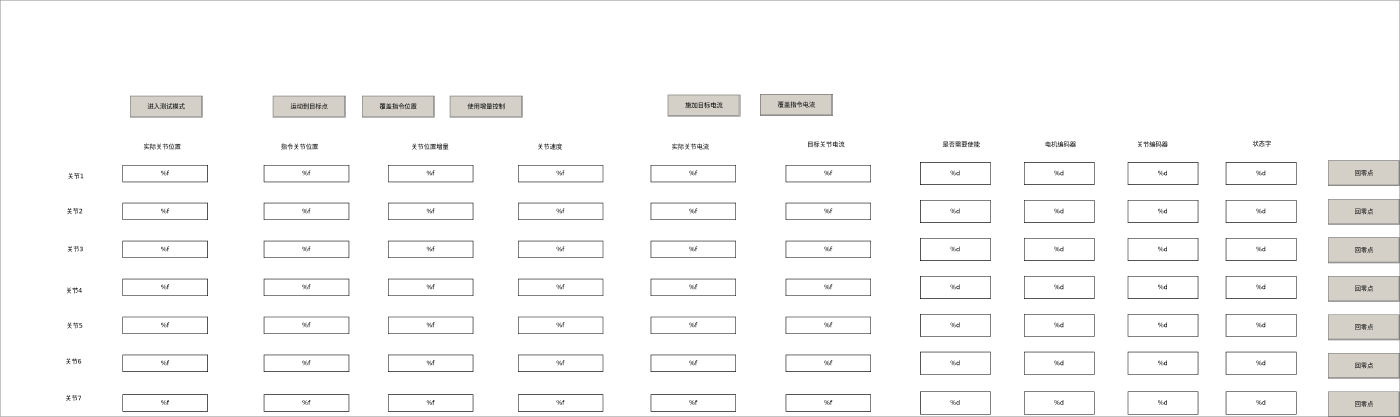
VISUALIZATION motion_a2  // 2468x736
    Label (211,244 150x30), "实际关节位置"
    Rectangle (216,291 150x30), "%f", text variable: g_motionTest.m_armDHJntPos[2][1]
    Label (453,244 150x30), "指令关节位置"
    Label (683,244 150x30), "关节位置增量"
    Rectangle (684,291 150x30), "%f", text variable: g_motionTest.m_targetJntPosInc[2][1]
        OnMouseClick: write the text variable via Default
    Label (1142,244 150x30), "实际关节电流"
    Rectangle (1147,291 150x30), "%f", text variable: g_motionTest.m_curJntCurrent[2][1]
    Label (1381,240 150x30), "目标关节电流"
    Rectangle (1385,291 150x30), "%f", text variable: g_motionTest.m_targetJntCurrent[2][1]
        OnMouseClick: write the text variable via Default
    Rectangle (216,358 150x30), "%f", text variable: g_motionTest.m_armDHJntPos[2][2]
    Rectangle (216,425 150x30), "%f", text variable: g_motionTest.m_armDHJntPos[2][3]
    Rectangle (216,492 150x30), "%f", text variable: g_motionTest.m_armDHJntPos[2][4]
    Rectangle (216,559 150x30), "%f", text variable: g_motionTest.m_armDHJntPos[2][5]
    Rectangle (216,626 150x30), "%f", text variable: g_motionTest.m_armDHJntPos[2][6]
    Rectangle (216,696 150x30), "%f", text variable: g_motionTest.m_armDHJntPos[2][7]
    Rectangle (465,291 150x30), "%f", text variable: g_motionTest.m_targetJntPos[2][1]
        OnMouseClick: write the text variable via Default
    Rectangle (465,358 150x30), "%f", text variable: g_motionTest.m_targetJntPos[2][2]
        OnMouseClick: write the text variable via Default
    Rectangle (465,425 150x30), "%f", text variable: g_motionTest.m_targetJntPos[2][3]
        OnMouseClick: write the text variable via Default
    Rectangle (465,492 150x30), "%f", text variable: g_motionTest.m_targetJntPos[2][4]
        OnMouseClick: write the text variable via Default
    Rectangle (465,559 150x30), "%f", text variable: g_motionTest.m_targetJntPos[2][5]
        OnMouseClick: write the text variable via Default
    Rectangle (465,626 150x30), "%f", text variable: g_motionTest.m_targetJntPos[2][6]
        OnMouseClick: write the text variable via Default
    Rectangle (465,696 150x30), "%f", text variable: g_motionTest.m_targetJntPos[2][7]
        OnMouseClick: write the text variable via Default
    Rectangle (684,358 150x30), "%f", text variable: g_motionTest.m_targetJntPosInc[2][2]
        OnMouseClick: write the text variable via Default
    Rectangle (684,425 150x30), "%f", text variable: g_motionTest.m_targetJntPosInc[2][3]
        OnMouseClick: write the text variable via Default
    Rectangle (684,492 150x30), "%f", text variable: g_motionTest.m_targetJntPosInc[2][4]
        OnMouseClick: write the text variable via Default
    Rectangle (684,559 150x30), "%f", text variable: g_motionTest.m_targetJntPosInc[2][5]
        OnMouseClick: write the text variable via Default
    Rectangle (684,626 150x30), "%f", text variable: g_motionTest.m_targetJntPosInc[2][6]
        OnMouseClick: write the text variable via Default
    Rectangle (684,696 150x30), "%f", text variable: g_motionTest.m_targetJntPosInc[2][7]
        OnMouseClick: write the text variable via Default
    Rectangle (1385,358 150x30), "%f", text variable: g_motionTest.m_targetJntCurrent[2][2]
        OnMouseClick: write the text variable via Default
    Rectangle (1385,425 150x30), "%f", text variable: g_motionTest.m_targetJntCurrent[2][3]
        OnMouseClick: write the text variable via Default
    Rectangle (1385,492 150x30), "%f", text variable: g_motionTest.m_targetJntCurrent[2][4]
        OnMouseClick: write the text variable via Default
    Rectangle (1385,559 150x30), "%f", text variable: g_motionTest.m_targetJntCurrent[2][5]
        OnMouseClick: write the text variable via Default
    Rectangle (1385,626 150x30), "%f", text variable: g_motionTest.m_targetJntCurrent[2][6]
        OnMouseClick: write the text variable via Default
    Rectangle (1385,696 150x30), "%f", text variable: g_motionTest.m_targetJntCurrent[2][7]
        OnMouseClick: write the text variable via Default
    Rectangle (1147,358 150x30), "%f", text variable: g_motionTest.m_curJntCurrent[2][2]
    Rectangle (1147,425 150x30), "%f", text variable: g_motionTest.m_curJntCurrent[2][3]
    Rectangle (1147,492 150x30), "%f", text variable: g_motionTest.m_curJntCurrent[2][4]
    Rectangle (1147,559 150x30), "%f", text variable: g_motionTest.m_curJntCurrent[2][5]
    Rectangle (1147,626 150x30), "%f", text variable: g_motionTest.m_curJntCurrent[2][6]
    Rectangle (1147,696 150x30), "%f", text variable: g_motionTest.m_curJntCurrent[2][7]
    Label (894,244 150x30), "关节速度"
    Rectangle (913,291 150x30), "%f", text variable: g_motionTest.m_targetJntVel[2][1]
        OnMouseClick: write the text variable via Default
    Rectangle (913,358 150x30), "%f", text variable: g_motionTest.m_targetJntVel[2][2]
        OnMouseClick: write the text variable via Default
    Rectangle (913,425 150x30), "%f", text variable: g_motionTest.m_targetJntVel[2][3]
        OnMouseClick: write the text variable via Default
    Rectangle (913,492 150x30), "%f", text variable: g_motionTest.m_targetJntVel[2][4]
        OnMouseClick: write the text variable via Default
    Rectangle (913,559 150x30), "%f", text variable: g_motionTest.m_targetJntVel[2][5]
        OnMouseClick: write the text variable via Default
    Rectangle (913,626 150x30), "%f", text variable: g_motionTest.m_targetJntVel[2][6]
        OnMouseClick: write the text variable via Default
    Rectangle (913,696 150x30), "%f", text variable: g_motionTest.m_targetJntVel[2][7]
        OnMouseClick: write the text variable via Default
    Button (229,169 128x38), "进入测试模式", colour toggle: g_motionTest.m_enterPrecisionTestMode[2]
        toggle g_motionTest.m_enterPrecisionTestMode[2]
    Button (481,169 128x38), "运动到目标点", colour toggle: g_motionTest.m_uiArmMode[2,1]
        tap g_motionTest.m_uiArmMode[2,1]
    Button (1177,167 128x38), "施加目标电流", colour toggle: g_motionTest.m_uiArmMode[2,8]
        toggle g_motionTest.m_uiArmMode[2,8]
    Button (793,169 128x38), "使用增量控制", colour toggle: g_motionTest.m_jntPosIncMode[2]
        toggle g_motionTest.m_jntPosIncMode[2]
    Label (1622,240 145x30), "是否需要使能"
    Rectangle (1622,286 124x40), "%d", text variable: g_motionTest.m_jntEnable[2][1]
        OnMouseClick: write the text variable via Default
    Rectangle (1622,353 124x40), "%d", text variable: g_motionTest.m_jntEnable[2][2]
        OnMouseClick: write the text variable via Default
    Rectangle (1622,420 124x40), "%d", text variable: g_motionTest.m_jntEnable[2][3]
        OnMouseClick: write the text variable via Default
    Rectangle (1622,487 124x40), "%d", text variable: g_motionTest.m_jntEnable[2][4]
        OnMouseClick: write the text variable via Default
    Rectangle (1622,554 124x40), "%d", text variable: g_motionTest.m_jntEnable[2][5]
        OnMouseClick: write the text variable via Default
    Rectangle (1622,621 124x40), "%d", text variable: g_motionTest.m_jntEnable[2][6]
        OnMouseClick: write the text variable via Default
    Rectangle (1622,691 124x40), "%d", text variable: g_motionTest.m_jntEnable[2][7]
        OnMouseClick: write the text variable via Default
    Label (1797,241 145x28), "电机编码器"
    Label (1959,241 145x28), "关节编码器"
    Label (2152,240 145x28), "状态字"
    Rectangle (1805,286 124x40), "%d", text variable: g_systemInfo.m_armJntInfo[2,1].m_motorInput.m_motorEncoder
    Rectangle (1805,353 124x40), "%d", text variable: g_systemInfo.m_armJntInfo[2,2].m_motorInput.m_motorEncoder
    Rectangle (1805,420 124x40), "%d", text variable: g_systemInfo.m_armJntInfo[2,3].m_motorInput.m_motorEncoder
    Rectangle (1805,487 124x40), "%d", text variable: g_systemInfo.m_armJntInfo[2,4].m_motorInput.m_motorEncoder
    Rectangle (1805,554 124x40), "%d", text variable: g_systemInfo.m_armJntInfo[2,5].m_motorInput.m_motorEncoder
    Rectangle (1805,621 124x40), "%d", text variable: g_systemInfo.m_armJntInfo[2,6].m_motorInput.m_motorEncoder
    Rectangle (1805,691 124x40), "%d", text variable: g_systemInfo.m_armJntInfo[2,7].m_motorInput.m_motorEncoder
    Rectangle (1988,286 124x40), "%d", text variable: g_systemInfo.m_armJntInfo[2,1].m_motorInput.m_linkEncoder
    Rectangle (1988,353 124x40), "%d", text variable: g_systemInfo.m_armJntInfo[2,2].m_motorInput.m_linkEncoder
    Rectangle (1988,420 124x40), "%d", text variable: g_systemInfo.m_armJntInfo[2,3].m_motorInput.m_linkEncoder
    Rectangle (1988,487 124x40), "%d", text variable: g_systemInfo.m_armJntInfo[2,4].m_motorInput.m_linkEncoder
    Rectangle (1988,554 124x40), "%d", text variable: g_systemInfo.m_armJntInfo[2,5].m_motorInput.m_linkEncoder
    Rectangle (1988,621 124x40), "%d", text variable: g_systemInfo.m_armJntInfo[2,6].m_motorInput.m_linkEncoder
    Rectangle (1988,691 124x40), "%d", text variable: g_systemInfo.m_armJntInfo[2,7].m_motorInput.m_linkEncoder
    Rectangle (2161,286 124x40), "%d", text variable: g_systemInfo.m_armJntInfo[2,1].m_motorInput.m_statusWord
    Rectangle (2161,353 124x40), "%d", text variable: g_systemInfo.m_armJntInfo[2,2].m_motorInput.m_statusWord
    Rectangle (2161,420 124x40), "%d", text variable: g_systemInfo.m_armJntInfo[2,3].m_motorInput.m_statusWord
    Rectangle (2161,487 124x40), "%d", text variable: g_systemInfo.m_armJntInfo[2,4].m_motorInput.m_statusWord
    Rectangle (2161,554 124x40), "%d", text variable: g_systemInfo.m_armJntInfo[2,5].m_motorInput.m_statusWord
    Rectangle (2161,621 124x40), "%d", text variable: g_systemInfo.m_armJntInfo[2,6].m_motorInput.m_statusWord
    Rectangle (2161,691 124x40), "%d", text variable: g_systemInfo.m_armJntInfo[2,7].m_motorInput.m_statusWord
    Button (638,169 128x38), "覆盖指令位置", colour toggle: g_motionTest.m_coverCmdPos[2]
        tap g_motionTest.m_coverCmdPos[2]
    Label (82,293 103x36), "关节1"
    Label (80,355 103x36), "关节2"
    Label (81,422 103x36), "关节3"
    Label (79,495 103x36), "关节4"
    Label (80,557 103x36), "关节5"
    Label (78,620 103x36), "关节6"
    Label (78,685 103x36), "关节7"
    Button (2341,283 127x45), "回零点", colour toggle: g_motionTest.m_goHome[2][1]
        tap g_motionTest.m_goHome[2][1]
    Button (2341,351 127x45), "回零点", colour toggle: g_motionTest.m_goHome[2][2]
        tap g_motionTest.m_goHome[2][2]
    Button (2341,419 127x45), "回零点", colour toggle: g_motionTest.m_goHome[2][3]
        tap g_motionTest.m_goHome[2][3]
    Button (2341,487 127x45), "回零点", colour toggle: g_motionTest.m_goHome[2][4]
        tap g_motionTest.m_goHome[2][4]
    Button (2341,555 127x45), "回零点", colour toggle: g_motionTest.m_goHome[2][5]
        tap g_motionTest.m_goHome[2][5]
    Button (2341,623 127x45), "回零点", colour toggle: g_motionTest.m_goHome[2][6]
        tap g_motionTest.m_goHome[2][6]
    Button (2341,691 127x45), "回零点", colour toggle: g_motionTest.m_goHome[2][7]
        tap g_motionTest.m_goHome[2][7]
    Button (1340,166 128x38), "覆盖指令电流", colour toggle: g_motionTest.m_coverCmdCurrent[2]
        tap g_motionTest.m_coverCmdCurrent[2]
END_VISUALIZATION

(* stored: Version 1.1.0.1, ProductVersion 3.1.4024.11
   Visu motion_a2: Id {2b420058-1a3b-41a3-a5ba-17830e6ad0ea} *)
